FUNCTION_BLOCK FB_ConsoleLogger IMPLEMENTS IEventLogger
VAR_INPUT
END_VAR
VAR_OUTPUT
	 sLastMessage : STRING(255);
END_VAR
VAR
END_VAR

{analysis 'TcLog'}
METHOD LogEvent : BOOL
VAR_INPUT
	sMessage	: STRING;
END_VAR
sLastMessage := sMessage;
LogEvent := TRUE; 

ADSLOGSTR(msgCtrlMask:= ADSLOG_MSGTYPE_HINT, msgFmtStr:= 'My log message: %s', strArg:= sMessage);
END_METHOD

END_FUNCTION_BLOCK

(* stored: Version 1.1.0.1
   POU FB_ConsoleLogger: Id {0be7e400-a2f1-4c7b-b343-c0d5d3a6bb1d}, SpecialFunc None
   Method LogEvent: Id {39b26e55-6806-449a-8dca-32cce5ddd8fb} *)
